positionExtrema := ruckig._profiles[1].positionExtrema();
AssertEquals_LREAL(0.13598633944686283614, positionExtrema.Tmax, 1E-9, message:='Profile[1] Tmax incorrect');
AssertEquals_LREAL(5.98711873384755755012, positionExtrema.Maximum, 1E-9, message:='Profile[1] maximum incorrect');
AssertEquals_LREAL(0.00000000000000000000, positionExtrema.Tmin, 1E-9, message:='Profile[1] Tmin incorrect');
AssertEquals_LREAL(-77.67370458831963730972, positionExtrema.Minimum, 1E-9, message:='Profile[1] minimum incorrect');

positionExtrema := ruckig._profiles[2].positionExtrema();
AssertEquals_LREAL(0.14901888909886754075, positionExtrema.Tmax, 1E-9, message:='Profile[2] Tmax incorrect');
AssertEquals_LREAL(92.98580498819549688960, positionExtrema.Maximum, 1E-9, message:='Profile[2] maximum incorrect');
AssertEquals_LREAL(0.00000000000000000000, positionExtrema.Tmin, 1E-9, message:='Profile[2] Tmin incorrect');
AssertEquals_LREAL(-11.76145133517785268396, positionExtrema.Minimum, 1E-9, message:='Profile[2] minimum incorrect');
   

TEST_FINISHED();
END_METHOD

METHOD Test_Trajectory_HasTargetVelocity_HasTargetAcceleration_41
VAR_INST
  ruckig : Struckig.Otg(0.001, 3) := (
  
    Synchronization := SynchronizationType.TimeSync,        
    MaxVelocity := [ 2000.00000000000000000000, 2000.00000000000000000000, 2000.00000000000000000000 ],
    MaxAcceleration := [ 20000.00000000000000000000, 20000.00000000000000000000, 20000.00000000000000000000 ],
    MaxJerk := [ 800000.00000000000000000000, 800000.00000000000000000000, 800000.00000000000000000000 ],
    CurrentPosition := [ 77.70133891525995295524, 7.01592092562633240505, 41.88398938907070601090 ],
    CurrentVelocity := [ -954.47536643469038608600, -572.16261829852851406031, 473.16402135503631143365 ],
    CurrentAcceleration := [ -2847.17654342300011194311, -1889.61698757276462856680, -3110.21768918452016805531 ],
    TargetPosition := [ 92.37579717709354554245, -14.04614057772144519731, -73.88361356505039623244 ],
    TargetVelocity := [ 519.95772801058456025203, 127.89327712966064609645, -380.91422286825297760515 ],
    TargetAcceleration := [ -890.64075852453197512659, 681.51569675393488978443, 390.99828361762297390669 ]
  );
  
  positionExtrema : Struckig.PositionExtremaDesc;
END_VAR
TEST('Trajectory_HasTargetVelocity_HasTargetAcceleration_41');

ruckig();

// Check total duration of profiles
AssertEquals_LREAL(Expected := 0.18543052523247699481, Actual := ruckig.Duration, DELTA := 1E-8, Message := 'Duration incorrect');

// Check duration for each phase
positionExtrema := ruckig._profiles[0].positionExtrema();
AssertEquals_LREAL(0.18543052523247699481, positionExtrema.Tmax, 1E-9, message:='Profile[0] Tmax incorrect');
AssertEquals_LREAL(92.37579717709354554245, positionExtrema.Maximum, 1E-9, message:='Profile[0] maximum incorrect');
AssertEquals_LREAL(0.07568410654937982041, positionExtrema.Tmin, 1E-9, message:='Profile[0] Tmin incorrect');
AssertEquals_LREAL(41.15768150995504015555, positionExtrema.Minimum, 1E-9, message:='Profile[0] minimum incorrect');

positionExtrema := ruckig._profiles[1].positionExtrema();
AssertEquals_LREAL(0.00000000000000000000, positionExtrema.Tmax, 1E-9, message:='Profile[1] Tmax incorrect');
AssertEquals_LREAL(7.01592092562633240505, positionExtrema.Maximum, 1E-9, message:='Profile[1] maximum incorrect');
AssertEquals_LREAL(0.16752625845292970497, positionExtrema.Tmin, 1E-9, message:='Profile[1] Tmin incorrect');
AssertEquals_LREAL(-15.47801998831725711625, positionExtrema.Minimum, 1E-9, message:='Profile[1] minimum incorrect');

positionExtrema := ruckig._profiles[2].positionExtrema();
AssertEquals_LREAL(0.02111222788851935261, positionExtrema.Tmax, 1E-9, message:='Profile[2] Tmax incorrect');
AssertEquals_LREAL(49.92568034606993876423, positionExtrema.Maximum, 1E-9, message:='Profile[2] maximum incorrect');
AssertEquals_LREAL(0.18543052523247699481, positionExtrema.Tmin, 1E-9, message:='Profile[2] Tmin incorrect');
AssertEquals_LREAL(-73.88361356505039623244, positionExtrema.Minimum, 1E-9, message:='Profile[2] minimum incorrect');
   

TEST_FINISHED();
END_METHOD

METHOD Test_Trajectory_HasTargetVelocity_HasTargetAcceleration_46
VAR_INST
  ruckig : Struckig.Otg(0.001, 3) := (
  
    Synchronization := SynchronizationType.TimeSync,        
    MaxVelocity := [ 2000.00000000000000000000, 2000.00000000000000000000, 2000.00000000000000000000 ],
    MaxAcceleration := [ 20000.00000000000000000000, 20000.00000000000000000000, 20000.00000000000000000000 ],
    MaxJerk := [ 800000.00000000000000000000, 800000.00000000000000000000, 800000.00000000000000000000 ],
    CurrentPosition := [ -81.70058267564624543411, -19.21897702137916041920, 94.53377990477645198553 ],
    CurrentVelocity := [ 791.96608977333426082623, 567.98007664216197554197, 949.19373974938935134560 ],
    CurrentAcceleration := [ -9852.41254141048739256803, -751.99368634466736693867, 3617.41551680202064744662 ],
    TargetPosition := [ 4.61526430014728816786, 47.19472748930556349478, -27.25527375543330776964 ],
    TargetVelocity := [ -365.39593288733976805815, -832.73312185042618693842, 15.48785727174674775597 ],
    TargetAcceleration := [ 393.54024330782590368472, -760.25458815149545444001, 23.06111995903222577908 ]
  );
  
  positionExtrema : Struckig.PositionExtremaDesc;
END_VAR
TEST('Trajectory_HasTargetVelocity_HasTargetAcceleration_46');

ruckig();

// Check total duration of profiles
AssertEquals_LREAL(Expected := 0.25941536116832880632, Actual := ruckig.Duration, DELTA := 1E-8, Message := 'Duration incorrect');

// Check duration for each phase
positionExtrema := ruckig._profiles[0].positionExtrema();
AssertEquals_LREAL(0.23392343586419403478, positionExtrema.Tmax, 1E-9, message:='Profile[0] Tmax incorrect');
AssertEquals_LREAL(11.84902844379517183881, positionExtrema.Maximum, 1E-9, message:='Profile[0] maximum incorrect');
AssertEquals_LREAL(0.00000000000000000000, positionExtrema.Tmin, 1E-9, message:='Profile[0] Tmin incorrect');
AssertEquals_LREAL(-81.70058267564624543411, positionExtrema.Minimum, 1E-9, message:='Profile[0] minimum incorrect');

positionExtrema := ruckig._profiles[1].positionExtrema();
AssertEquals_LREAL(0.19491405447314413824, positionExtrema.Tmax, 1E-9, message:='Profile[1] Tmax incorrect');
AssertEquals_LREAL(72.37093782213797510394, positionExtrema.Maximum, 1E-9, message:='Profile[1] maximum incorrect');
AssertEquals_LREAL(0.00000000000000000000, positionExtrema.Tmin, 1E-9, message:='Profile[1] Tmin incorrect');
AssertEquals_LREAL(-19.21897702137916041920, positionExtrema.Minimum, 1E-9, message:='Profile[1] minimum incorrect');

positionExtrema := ruckig._profiles[2].positionExtrema();
AssertEquals_LREAL(0.02952176939600252917, positionExtrema.Tmax, 1E-9, message:='Profile[2] Tmax incorrect');
AssertEquals_LREAL(120.70144362619019773319, positionExtrema.Maximum, 1E-9, message:='Profile[2] maximum incorrect');
AssertEquals_LREAL(0.25322160979530433655, positionExtrema.Tmin, 1E-9, message:='Profile[2] Tmin incorrect');
AssertEquals_LREAL(-27.31907826634350300310, positionExtrema.Minimum, 1E-9, message:='Profile[2] minimum incorrect');
   

TEST_FINISHED();
END_METHOD

METHOD Test_Trajectory_HasTargetVelocity_HasTargetAcceleration_47
VAR_INST
  ruckig : Struckig.Otg(0.001, 3) := (
  
    Synchronization := SynchronizationType.TimeSync,        
    MaxVelocity := [ 2000.00000000000000000000, 2000.00000000000000000000, 2000.00000000000000000000 ],
    MaxAcceleration := [ 20000.00000000000000000000, 20000.00000000000000000000, 20000.00000000000000000000 ],
    MaxJerk := [ 800000.00000000000000000000, 800000.00000000000000000000, 800000.00000000000000000000 ],
    CurrentPosition := [ 81.61368863479273727535, 18.81647567172932156154, -89.15971183512543518646 ],
    CurrentVelocity := [ 614.05723536338791745948, 343.05287387529847364931, -371.00163086153361291508 ],
    CurrentAcceleration := [ 2762.36060607538092881441, -8252.84383845068077789620, 1522.48694311787949118298 ],
    TargetPosition := [ 31.53792392446635517445, -13.15393306556988761713, -67.81554985684867631335 ],
    TargetVelocity := [ 927.36256285251761255495, -453.39442766394324735302, -734.53754957298599492788 ],
    TargetAcceleration := [ -810.42747656261008160072, 683.82844872197824770410, -296.63416710646515639382 ]
  );
  
  positionExtrema : Struckig.PositionExtremaDesc;
END_VAR
TEST('Trajectory_HasTargetVelocity_HasTargetAcceleration_47');

ruckig();

// Check total duration of profiles
AssertEquals_LREAL(Expected := 0.25287606970423076591, Actual := ruckig.Duration, DELTA := 1E-8, Message := 'Duration incorrect');

// Check duration for each phase
positionExtrema := ruckig._profiles[0].positionExtrema();
AssertEquals_LREAL(0.02845295075759422462, positionExtrema.Tmax, 1E-9, message:='Profile[0] Tmax incorrect');
AssertEquals_LREAL(97.13230269209392986340, positionExtrema.Maximum, 1E-9, message:='Profile[0] maximum incorrect');
AssertEquals_LREAL(0.22686303535852750390, positionExtrema.Tmin, 1E-9, message:='Profile[0] Tmin incorrect');
AssertEquals_LREAL(9.48720344289291794837, positionExtrema.Minimum, 1E-9, message:='Profile[0] minimum incorrect');

positionExtrema := ruckig._profiles[1].positionExtrema();
AssertEquals_LREAL(0.02241468542399701822, positionExtrema.Tmax, 1E-9, message:='Profile[1] Tmax incorrect');
AssertEquals_LREAL(23.03639977720293785524, positionExtrema.Maximum, 1E-9, message:='Profile[1] maximum incorrect');
AssertEquals_LREAL(0.25287606970423076591, positionExtrema.Tmin, 1E-9, message:='Profile[1] Tmin incorrect');
AssertEquals_LREAL(-13.15393306556988761713, positionExtrema.Minimum, 1E-9, message:='Profile[1] minimum incorrect');

positionExtrema := ruckig._profiles[2].positionExtrema();
AssertEquals_LREAL(0.20039624088411220337, positionExtrema.Tmax, 1E-9, message:='Profile[2] Tmax incorrect');
AssertEquals_LREAL(-46.06681198459425274905, positionExtrema.Maximum, 1E-9, message:='Profile[2] maximum incorrect');
AssertEquals_LREAL(0.03284040362274634473, positionExtrema.Tmin, 1E-9, message:='Profile[2] Tmin incorrect');
AssertEquals_LREAL(-95.92347928545005686374, positionExtrema.Minimum, 1E-9, message:='Profile[2] minimum incorrect');
   

TEST_FINISHED();
END_METHOD

METHOD Test_Trajectory_HasTargetVelocity_HasTargetAcceleration_48
VAR_INST
  ruckig : Struckig.Otg(0.001, 3) := (
  
    Synchronization := SynchronizationType.TimeSync,        
    MaxVelocity := [ 2000.00000000000000000000, 2000.00000000000000000000, 2000.00000000000000000000 ],
    MaxAcceleration := [ 20000.00000000000000000000, 20000.00000000000000000000, 20000.00000000000000000000 ],
    MaxJerk := [ 800000.00000000000000000000, 800000.00000000000000000000, 800000.00000000000000000000 ],
    CurrentPosition := [ -88.66208591478776668282, -31.58880789945652622919, 65.04291982806716987398 ],
    CurrentVelocity := [ 580.03497340359649570019, -746.36896556027750193607, 812.20588456619907447021 ],
    CurrentAcceleration := [ -6519.58462448879436124116, -9252.12079111587627266999, -5505.83185145304014440626 ],
    TargetPosition := [ -85.04127215306982634502, -92.28954144915404356198, -74.37698578032075147348 ],
    TargetVelocity := [ -365.82662455999411577068, -112.69189210154274860543, 154.77689249662125803297 ],
    TargetAcceleration := [ -682.87003825383567345852, -247.18670592987155032461, -122.60845320130738400621 ]
  );
  
  positionExtrema : Struckig.PositionExtremaDesc;
END_VAR
TEST('Trajectory_HasTargetVelocity_HasTargetAcceleration_48');

ruckig();

// Check total duration of profiles
AssertEquals_LREAL(Expected := 0.25037129752792702808, Actual := ruckig.Duration, DELTA := 1E-8, Message := 'Duration incorrect');

// Check duration for each phase
positionExtrema := ruckig._profiles[0].positionExtrema();
AssertEquals_LREAL(0.04415928948418586242, positionExtrema.Tmax, 1E-9, message:='Profile[0] Tmax incorrect');
AssertEquals_LREAL(-76.79539758143890537667, positionExtrema.Maximum, 1E-9, message:='Profile[0] maximum incorrect');
AssertEquals_LREAL(0.00000000000000000000, positionExtrema.Tmin, 1E-9, message:='Profile[0] Tmin incorrect');
AssertEquals_LREAL(-88.66208591478776668282, positionExtrema.Minimum, 1E-9, message:='Profile[0] minimum incorrect');

positionExtrema := ruckig._profiles[1].positionExtrema();
AssertEquals_LREAL(0.00000000000000000000, positionExtrema.Tmax, 1E-9, message:='Profile[1] Tmax incorrect');
AssertEquals_LREAL(-31.58880789945652622919, positionExtrema.Maximum, 1E-9, message:='Profile[1] maximum incorrect');
AssertEquals_LREAL(0.25037129752792697257, positionExtrema.Tmin, 1E-9, message:='Profile[1] Tmin incorrect');
AssertEquals_LREAL(-92.28954144915404356198, positionExtrema.Minimum, 1E-9, message:='Profile[1] minimum incorrect');

positionExtrema := ruckig._profiles[2].positionExtrema();
AssertEquals_LREAL(0.01811771018568369973, positionExtrema.Tmax, 1E-9, message:='Profile[2] Tmax incorrect');
AssertEquals_LREAL(78.06162686897538094399, positionExtrema.Maximum, 1E-9, message:='Profile[2] maximum incorrect');
AssertEquals_LREAL(0.23054659268189173216, positionExtrema.Tmin, 1E-9, message:='Profile[2] Tmin incorrect');
AssertEquals_LREAL(-76.43062116116439597135, positionExtrema.Minimum, 1E-9, message:='Profile[2] minimum incorrect');
   

TEST_FINISHED();
END_METHOD

METHOD Test_Trajectory_HasTargetVelocity_HasTargetAcceleration_51
VAR_INST
  ruckig : Struckig.Otg(0.001, 3) := (
  
    Synchronization := SynchronizationType.TimeSync,        
    MaxVelocity := [ 2000.00000000000000000000, 2000.00000000000000000000, 2000.00000000000000000000 ],
    MaxAcceleration := [ 20000.00000000000000000000, 20000.00000000000000000000, 20000.00000000000000000000 ],
    MaxJerk := [ 800000.00000000000000000000, 800000.00000000000000000000, 800000.00000000000000000000 ],
    CurrentPosition := [ 52.80919631150752024951, -81.68038555889982887948, 42.06917442755320735159 ],
    CurrentVelocity := [ -848.38044536898496517097, -694.53443230755419790512, -67.27027959540748724976 ],
    CurrentAcceleration := [ -7839.42279939661148091545, 2086.65454098016925854608, -1769.91408787331420171540 ],
    TargetPosition := [ 18.36498902426966139956, 7.18108207234031681310, -24.86667965964299753523 ],
    TargetVelocity := [ -484.52530887106502177630, -330.54249305132475456048, 184.78707869201707580942 ],
    TargetAcceleration := [ 34.47472473095945133537, 524.15868234202798703336, 659.72269096659351816925 ]
  );
  
  positionExtrema : Struckig.PositionExtremaDesc;
END_VAR
TEST('Trajectory_HasTargetVelocity_HasTargetAcceleration_51');

ruckig();

// Check total duration of profiles
AssertEquals_LREAL(Expected := 0.22814955969060143892, Actual := ruckig.Duration, DELTA := 1E-8, Message := 'Duration incorrect');

// Check duration for each phase
positionExtrema := ruckig._profiles[0].positionExtrema();
AssertEquals_LREAL(0.00000000000000000000, positionExtrema.Tmax, 1E-9, message:='Profile[0] Tmax incorrect');
AssertEquals_LREAL(52.80919631150752024951, positionExtrema.Maximum, 1E-9, message:='Profile[0] maximum incorrect');
AssertEquals_LREAL(0.06738171645932469755, positionExtrema.Tmin, 1E-9, message:='Profile[0] Tmin incorrect');
AssertEquals_LREAL(13.99608603958429142722, positionExtrema.Minimum, 1E-9, message:='Profile[0] minimum incorrect');

positionExtrema := ruckig._profiles[1].positionExtrema();
AssertEquals_LREAL(0.20249436133767390045, positionExtrema.Tmax, 1E-9, message:='Profile[1] Tmax incorrect');
AssertEquals_LREAL(13.58224981559266097975, positionExtrema.Maximum, 1E-9, message:='Profile[1] maximum incorrect');
AssertEquals_LREAL(0.02239168182377478805, positionExtrema.Tmin, 1E-9, message:='Profile[1] Tmin incorrect');
AssertEquals_LREAL(-95.21214742443424938756, positionExtrema.Minimum, 1E-9, message:='Profile[1] minimum incorrect');

positionExtrema := ruckig._profiles[2].positionExtrema();
AssertEquals_LREAL(0.00000000000000000000, positionExtrema.Tmax, 1E-9, message:='Profile[2] Tmax incorrect');
AssertEquals_LREAL(42.06917442755320735159, positionExtrema.Maximum, 1E-9, message:='Profile[2] maximum incorrect');
AssertEquals_LREAL(0.20746496504559683305, positionExtrema.Tmin, 1E-9, message:='Profile[2] Tmin incorrect');
AssertEquals_LREAL(-27.36779954300167716497, positionExtrema.Minimum, 1E-9, message:='Profile[2] minimum incorrect');
   

TEST_FINISHED();
END_METHOD

METHOD Test_Trajectory_HasTargetVelocity_HasTargetAcceleration_56
VAR_INST
  ruckig : Struckig.Otg(0.001, 3) := (
  
    Synchronization := SynchronizationType.TimeSync,        
    MaxVelocity := [ 2000.00000000000000000000, 2000.00000000000000000000, 2000.00000000000000000000 ],
    MaxAcceleration := [ 20000.00000000000000000000, 20000.00000000000000000000, 20000.00000000000000000000 ],
    MaxJerk := [ 800000.00000000000000000000, 800000.00000000000000000000, 800000.00000000000000000000 ],
    CurrentPosition := [ -75.10494070961726720270, -6.22395011546019816251, 35.64048680664691914899 ],
    CurrentVelocity := [ -825.41867748520257919154, -559.17669137031361970003, 331.05712850319173412572 ],
    CurrentAcceleration := [ -2748.49249899548522080295, -2734.78689775577458931366, 8828.96129221495357342064 ],
    TargetPosition := [ -88.93249178580995817356, 32.61549251092765189242, -4.33333209618611192582 ],
    TargetVelocity := [ -969.86803709259822880995, 219.52159207481986413768, 145.45315840784223837545 ],
    TargetAcceleration := [ 673.73439439858611876843, 589.54870253816602598818, 268.61037017006333371683 ]
  );
  
  positionExtrema : Struckig.PositionExtremaDesc;
END_VAR
TEST('Trajectory_HasTargetVelocity_HasTargetAcceleration_56');

ruckig();

// Check total duration of profiles
AssertEquals_LREAL(Expected := 0.22533279528439006945, Actual := ruckig.Duration, DELTA := 1E-8, Message := 'Duration incorrect');

// Check duration for each phase
positionExtrema := ruckig._profiles[0].positionExtrema();
AssertEquals_LREAL(0.13546282954524005437, positionExtrema.Tmax, 1E-9, message:='Profile[0] Tmax incorrect');
AssertEquals_LREAL(-60.83093977470542768060, positionExtrema.Maximum, 1E-9, message:='Profile[0] maximum incorrect');
AssertEquals_LREAL(0.08546282954524006548, positionExtrema.Tmin, 1E-9, message:='Profile[0] Tmin incorrect');
AssertEquals_LREAL(-97.18448406099201974939, positionExtrema.Minimum, 1E-9, message:='Profile[0] minimum incorrect');

positionExtrema := ruckig._profiles[1].positionExtrema();
AssertEquals_LREAL(0.22533279528439004169, positionExtrema.Tmax, 1E-9, message:='Profile[1] Tmax incorrect');
AssertEquals_LREAL(32.61549251092765189242, positionExtrema.Maximum, 1E-9, message:='Profile[1] maximum incorrect');
AssertEquals_LREAL(0.04813186201257521613, positionExtrema.Tmin, 1E-9, message:='Profile[1] Tmin incorrect');
AssertEquals_LREAL(-22.45997635018479243740, positionExtrema.Minimum, 1E-9, message:='Profile[1] minimum incorrect');

positionExtrema := ruckig._profiles[2].positionExtrema();
AssertEquals_LREAL(0.04893648758049205100, positionExtrema.Tmax, 1E-9, message:='Profile[2] Tmax incorrect');
AssertEquals_LREAL(47.07359821757206930215, positionExtrema.Maximum, 1E-9, message:='Profile[2] maximum incorrect');
AssertEquals_LREAL(0.20659644161609555524, positionExtrema.Tmin, 1E-9, message:='Profile[2] Tmin incorrect');
AssertEquals_LREAL(-6.13445732070238047839, positionExtrema.Minimum, 1E-9, message:='Profile[2] minimum incorrect');
   

TEST_FINISHED();
END_METHOD

METHOD Test_Trajectory_HasTargetVelocity_HasTargetAcceleration_60
VAR_INST
  ruckig : Struckig.Otg(0.001, 3) := (
  
    Synchronization := SynchronizationType.TimeSync,        
    MaxVelocity := [ 2000.00000000000000000000, 2000.00000000000000000000, 2000.00000000000000000000 ],
    MaxAcceleration := [ 20000.00000000000000000000, 20000.00000000000000000000, 20000.00000000000000000000 ],
    MaxJerk := [ 800000.00000000000000000000, 800000.00000000000000000000, 800000.00000000000000000000 ],
    CurrentPosition := [ -82.30425131320278353542, 95.77277574475397159404, -0.37873053404373990816 ],
    CurrentVelocity := [ 209.81667767709768668283, 666.24835564548857291811, -156.12978395261052355636 ],
    CurrentAcceleration := [ 554.62083613543836690951, 1781.55274365866716834716, -2304.74829583103382901754 ],
    TargetPosition := [ 78.56604956044506593571, -99.70839917358892989796, -88.26279812419441839211 ],
    TargetVelocity := [ 182.35588906091311400814, 216.59536701599199659540, -100.01197301996137412061 ],
    TargetAcceleration := [ 165.30880475002527418837, -915.29760737648621216067, 984.89234990536533587147 ]
  );
  
  positionExtrema : Struckig.PositionExtremaDesc;
END_VAR
TEST('Trajectory_HasTargetVelocity_HasTargetAcceleration_60');

ruckig();

// Check total duration of profiles
AssertEquals_LREAL(Expected := 0.28418047012119368455, Actual := ruckig.Duration, DELTA := 1E-8, Message := 'Duration incorrect');

// Check duration for each phase
positionExtrema := ruckig._profiles[0].positionExtrema();
AssertEquals_LREAL(0.28418047012119368455, positionExtrema.Tmax, 1E-9, message:='Profile[0] Tmax incorrect');
AssertEquals_LREAL(78.56604956044506593571, positionExtrema.Maximum, 1E-9, message:='Profile[0] maximum incorrect');
AssertEquals_LREAL(0.00000000000000000000, positionExtrema.Tmin, 1E-9, message:='Profile[0] Tmin incorrect');
AssertEquals_LREAL(-82.30425131320278353542, positionExtrema.Minimum, 1E-9, message:='Profile[0] minimum incorrect');

positionExtrema := ruckig._profiles[1].positionExtrema();
AssertEquals_LREAL(0.02722694092957333306, positionExtrema.Tmax, 1E-9, message:='Profile[1] Tmax incorrect');
AssertEquals_LREAL(111.88188475863630344520, positionExtrema.Maximum, 1E-9, message:='Profile[1] maximum incorrect');
AssertEquals_LREAL(0.25973833461914580534, positionExtrema.Tmin, 1E-9, message:='Profile[1] Tmin incorrect');
AssertEquals_LREAL(-103.32890392255741573990, positionExtrema.Minimum, 1E-9, message:='Profile[1] minimum incorrect');

positionExtrema := ruckig._profiles[2].positionExtrema();
AssertEquals_LREAL(0.00000000000000000000, positionExtrema.Tmax, 1E-9, message:='Profile[2] Tmax incorrect');
AssertEquals_LREAL(-0.37873053404373990816, positionExtrema.Maximum, 1E-9, message:='Profile[2] maximum incorrect');
AssertEquals_LREAL(0.28418047012119368455, positionExtrema.Tmin, 1E-9, message:='Profile[2] Tmin incorrect');
AssertEquals_LREAL(-88.26279812419441839211, positionExtrema.Minimum, 1E-9, message:='Profile[2] minimum incorrect');
   

TEST_FINISHED();
END_METHOD

METHOD Test_Trajectory_HasTargetVelocity_HasTargetAcceleration_61
VAR_INST
  ruckig : Struckig.Otg(0.001, 3) := (
  
    Synchronization := SynchronizationType.TimeSync,        
    MaxVelocity := [ 2000.00000000000000000000, 2000.00000000000000000000, 2000.00000000000000000000 ],
    MaxAcceleration := [ 20000.00000000000000000000, 20000.00000000000000000000, 20000.00000000000000000000 ],
    MaxJerk := [ 800000.00000000000000000000, 800000.00000000000000000000, 800000.00000000000000000000 ],
    CurrentPosition := [ 69.02958196301639759440, -13.39780118806328346182, -96.66107573544628905893 ],
    CurrentVelocity := [ 100.84225227141041614232, -40.44627894454811212199, 363.36834103503497317433 ],
    CurrentAcceleration := [ -7135.55942272971151396632, -622.60760459453013027087, 1671.34292984182866348419 ],
    TargetPosition := [ -16.84074689714994121914, -92.09682308688789476037, -87.06215904519353898650 ],
    TargetVelocity := [ 537.25106843782555188227, -935.18562117857493376505, -396.85249080038204283483 ],
    TargetAcceleration := [ -310.44042758873558796040, -501.02391325450025760802, -57.28028759093501776078 ]
  );
  
  positionExtrema : Struckig.PositionExtremaDesc;
END_VAR
TEST('Trajectory_HasTargetVelocity_HasTargetAcceleration_61');

ruckig();

// Check total duration of profiles
AssertEquals_LREAL(Expected := 0.19429164835544748824, Actual := ruckig.Duration, DELTA := 1E-8, Message := 'Duration incorrect');

// Check duration for each phase
positionExtrema := ruckig._profiles[0].positionExtrema();
AssertEquals_LREAL(0.00929214609675180735, positionExtrema.Tmax, 1E-9, message:='Profile[0] Tmax incorrect');
AssertEquals_LREAL(69.55159049131329140891, positionExtrema.Maximum, 1E-9, message:='Profile[0] maximum incorrect');
AssertEquals_LREAL(0.16890359782096156516, positionExtrema.Tmin, 1E-9, message:='Profile[0] Tmin incorrect');
AssertEquals_LREAL(-28.39869225356863324805, positionExtrema.Minimum, 1E-9, message:='Profile[0] minimum incorrect');

positionExtrema := ruckig._profiles[1].positionExtrema();
AssertEquals_LREAL(0.00000000000000000000, positionExtrema.Tmax, 1E-9, message:='Profile[1] Tmax incorrect');
AssertEquals_LREAL(-13.39780118806328346182, positionExtrema.Maximum, 1E-9, message:='Profile[1] maximum incorrect');
AssertEquals_LREAL(0.19429164835544748824, positionExtrema.Tmin, 1E-9, message:='Profile[1] Tmin incorrect');
AssertEquals_LREAL(-92.09682308688789476037, positionExtrema.Minimum, 1E-9, message:='Profile[1] minimum incorrect');

positionExtrema := ruckig._profiles[2].positionExtrema();
AssertEquals_LREAL(0.15958331587242960414, positionExtrema.Tmax, 1E-9, message:='Profile[2] Tmax incorrect');
AssertEquals_LREAL(-78.59507311744690127853, positionExtrema.Maximum, 1E-9, message:='Profile[2] maximum incorrect');
AssertEquals_LREAL(0.00000000000000000000, positionExtrema.Tmin, 1E-9, message:='Profile[2] Tmin incorrect');
AssertEquals_LREAL(-96.66107573544628905893, positionExtrema.Minimum, 1E-9, message:='Profile[2] minimum incorrect');
   

TEST_FINISHED();
END_METHOD

METHOD Test_Trajectory_HasTargetVelocity_HasTargetAcceleration_66
VAR_INST
  ruckig : Struckig.Otg(0.001, 3) := (
  
    Synchronization := SynchronizationType.TimeSync,        
    MaxVelocity := [ 2000.00000000000000000000, 2000.00000000000000000000, 2000.00000000000000000000 ],
    MaxAcceleration := [ 20000.00000000000000000000, 20000.00000000000000000000, 20000.00000000000000000000 ],
    MaxJerk := [ 800000.00000000000000000000, 800000.00000000000000000000, 800000.00000000000000000000 ],
    CurrentPosition := [ -48.80987185641822634352, 18.04364910313265113473, -24.74266082352920648191 ],
    CurrentVelocity := [ 988.42910759631240580347, -768.41448219800986407790, -207.75563249912386254437 ],
    CurrentAcceleration := [ 3735.71066306482680374756, -9295.98081225150599493645, 5866.28306601172880618833 ],
    TargetPosition := [ -12.17413972252995790768, 39.46835789725682275275, -82.53347662682273266910 ],
    TargetVelocity := [ 196.90336440418968777522, 718.33687283187941829965, -527.62167018153525077651 ],
    TargetAcceleration := [ -832.60782943610661277489, 502.29848616551748818893, 413.82241950646152872650 ]
  );
  
  positionExtrema : Struckig.PositionExtremaDesc;
END_VAR
TEST('Trajectory_HasTargetVelocity_HasTargetAcceleration_66');

ruckig();

// Check total duration of profiles
AssertEquals_LREAL(Expected := 0.15504630751390929833, Actual := ruckig.Duration, DELTA := 1E-8, Message := 'Duration incorrect');

// Check duration for each phase
positionExtrema := ruckig._profiles[0].positionExtrema();
AssertEquals_LREAL(0.06757881268766546823, positionExtrema.Tmax, 1E-9, message:='Profile[0] Tmax incorrect');
AssertEquals_LREAL(-7.34951569385982939053, positionExtrema.Maximum, 1E-9, message:='Profile[0] maximum incorrect');
AssertEquals_LREAL(0.00000000000000000000, positionExtrema.Tmin, 1E-9, message:='Profile[0] Tmin incorrect');
AssertEquals_LREAL(-48.80987185641822634352, positionExtrema.Minimum, 1E-9, message:='Profile[0] minimum incorrect');

positionExtrema := ruckig._profiles[1].positionExtrema();
AssertEquals_LREAL(0.15504630751390929833, positionExtrema.Tmax, 1E-9, message:='Profile[1] Tmax incorrect');
AssertEquals_LREAL(39.46835789725682275275, positionExtrema.Maximum, 1E-9, message:='Profile[1] maximum incorrect');
AssertEquals_LREAL(0.03661997601531438024, positionExtrema.Tmin, 1E-9, message:='Profile[1] Tmin incorrect');
AssertEquals_LREAL(-9.78096891406795521107, positionExtrema.Minimum, 1E-9, message:='Profile[1] minimum incorrect');

positionExtrema := ruckig._profiles[2].positionExtrema();
AssertEquals_LREAL(0.00000000000000000000, positionExtrema.Tmax, 1E-9, message:='Profile[2] Tmax incorrect');
AssertEquals_LREAL(-24.74266082352920648191, positionExtrema.Maximum, 1E-9, message:='Profile[2] maximum incorrect');
AssertEquals_LREAL(0.15504630751390929833, positionExtrema.Tmin, 1E-9, message:='Profile[2] Tmin incorrect');
AssertEquals_LREAL(-82.53347662682273266910, positionExtrema.Minimum, 1E-9, message:='Profile[2] minimum incorrect');
   

TEST_FINISHED();
END_METHOD

METHOD Test_Trajectory_HasTargetVelocity_HasTargetAcceleration_70
VAR_INST
  ruckig : Struckig.Otg(0.001, 3) := (
  
    Synchronization := SynchronizationType.TimeSync,        
    MaxVelocity := [ 2000.00000000000000000000, 2000.00000000000000000000, 2000.00000000000000000000 ],
    MaxAcceleration := [ 20000.00000000000000000000, 20000.00000000000000000000, 20000.00000000000000000000 ],
    MaxJerk := [ 800000.00000000000000000000, 800000.00000000000000000000, 800000.00000000000000000000 ],
    CurrentPosition := [ -92.33184858939047501281, 71.73781926022004995502, -55.27032026177170109804 ],
    CurrentVelocity := [ -952.87828015244156176777, -234.88833123485505893768, 123.27287252024666486250 ],
    CurrentAcceleration := [ -7266.87319497806674917229, -1917.48167665642540669069, -9579.01136324118306220043 ],
    TargetPosition := [ -64.62381428735777433303, 58.03768693667834099870, 63.08437907080863737974 ],
    TargetVelocity := [ 812.70256182329512739670, -863.39780178803880517080, -492.22548367060147711527 ],
    TargetAcceleration := [ 53.46404855095147468091, -729.77327604858464837889, -373.83030360848226791859 ]
  );
  
  positionExtrema : Struckig.PositionExtremaDesc;
END_VAR
TEST('Trajectory_HasTargetVelocity_HasTargetAcceleration_70');

ruckig();

// Check total duration of profiles
AssertEquals_LREAL(Expected := 0.22013991649512543169, Actual := ruckig.Duration, DELTA := 1E-8, Message := 'Duration incorrect');

// Check duration for each phase
positionExtrema := ruckig._profiles[0].positionExtrema();
AssertEquals_LREAL(0.22013991649512543169, positionExtrema.Tmax, 1E-9, message:='Profile[0] Tmax incorrect');
AssertEquals_LREAL(-64.62381428735777433303, positionExtrema.Maximum, 1E-9, message:='Profile[0] maximum incorrect');
AssertEquals_LREAL(0.08266151031223724355, positionExtrema.Tmin, 1E-9, message:='Profile[0] Tmin incorrect');
AssertEquals_LREAL(-135.90053229571682891219, positionExtrema.Minimum, 1E-9, message:='Profile[0] minimum incorrect');

positionExtrema := ruckig._profiles[1].positionExtrema();
AssertEquals_LREAL(0.16474949862477941687, positionExtrema.Tmax, 1E-9, message:='Profile[1] Tmax incorrect');
AssertEquals_LREAL(86.19544571063090643293, positionExtrema.Maximum, 1E-9, message:='Profile[1] maximum incorrect');
AssertEquals_LREAL(0.22013991649512543169, positionExtrema.Tmin, 1E-9, message:='Profile[1] Tmin incorrect');
AssertEquals_LREAL(58.03768693667834099870, positionExtrema.Minimum, 1E-9, message:='Profile[1] minimum incorrect');

positionExtrema := ruckig._profiles[2].positionExtrema();
AssertEquals_LREAL(0.19560720437463602339, positionExtrema.Tmax, 1E-9, message:='Profile[2] Tmax incorrect');
AssertEquals_LREAL(73.07882819675037922025, positionExtrema.Maximum, 1E-9, message:='Profile[2] maximum incorrect');
AssertEquals_LREAL(0.00000000000000000000, positionExtrema.Tmin, 1E-9, message:='Profile[2] Tmin incorrect');
AssertEquals_LREAL(-55.27032026177170109804, positionExtrema.Minimum, 1E-9, message:='Profile[2] minimum incorrect');
   

TEST_FINISHED();
END_METHOD

END_FUNCTION_BLOCK

// ---- POUs/PropagateTest.TcPOU
FUNCTION_BLOCK PropagateTest EXTENDS TcUnit.FB_TestSuite

Test_AutoPropagate();
Test_ManualPropagate();
Test_NoPropagate();

METHOD Test_AutoPropagate
VAR_INST
  ruckig : Struckig.Otg(0.001, 3) := (
  
    Synchronization := SynchronizationType.TimeSync,        
    MaxVelocity := [ 2000, 2000, 2000 ],
    MaxAcceleration := [ 20000, 20000, 20000 ],
    MaxJerk := [ 8000, 80000, 800000 ],
    CurrentPosition := [ 0,0,0  ],
    CurrentVelocity := [ 0,0,0 ],
    CurrentAcceleration := [ 0,0,0 ],
    TargetPosition := [ 1, 10, 100 ],
    TargetVelocity := [ 0,0,0 ],
    TargetAcceleration := [ 0,0,0 ]
  );
  
  StartPosition, StartVelocity, StartAcceleration : ARRAY[0..ParameterList.MaxDoFs] OF LREAL; // Current state
  NewPosition, NewVelocity, NewAcceleration : ARRAY[0..ParameterList.MaxDoFs] OF LREAL; // Current state  
END_VAR
TEST('Test_AutoPropagate');

StartPosition := ruckig.CurrentPosition;
StartVelocity := ruckig.CurrentVelocity;
StartAcceleration := ruckig.CurrentAcceleration;

ruckig();
AssertTrue(0 = ruckig.CurrentPosition[0], Message:=''); 

NewPosition := ruckig.NewPosition;
NewVelocity := ruckig.NewVelocity;
NewAcceleration := ruckig.NewAcceleration;

ruckig(EnableAutoPropagate := TRUE);

AssertTrue(0 <> ruckig.CurrentPosition[0], Message:=''); 
AssertArrayEquals_LREAL(Expecteds:=NewPosition, Actuals:=ruckig.CurrentPosition, Delta:=1E-6, Message:='');
AssertArrayEquals_LREAL(Expecteds:=NewVelocity, Actuals:=ruckig.CurrentVelocity, Delta:=1E-6, Message:='');
AssertArrayEquals_LREAL(Expecteds:=NewAcceleration, Actuals:=ruckig.CurrentAcceleration, Delta:=1E-6, Message:='');

TEST_FINISHED();
END_METHOD

METHOD Test_ManualPropagate
VAR_INST
  ruckig : Struckig.Otg(0.001, 3) := (
  
    Synchronization := SynchronizationType.TimeSync,        
    MaxVelocity := [ 2000, 2000, 2000 ],
    MaxAcceleration := [ 20000, 20000, 20000 ],
    MaxJerk := [ 8000, 80000, 800000 ],
    CurrentPosition := [ 0,0,0  ],
    CurrentVelocity := [ 0,0,0 ],
    CurrentAcceleration := [ 0,0,0 ],
    TargetPosition := [ 1, 10, 100 ],
    TargetVelocity := [ 0,0,0 ],
    TargetAcceleration := [ 0,0,0 ]
  );
  
  StartPosition, StartVelocity, StartAcceleration : ARRAY[0..ParameterList.MaxDoFs] OF LREAL; // Current state
  NewPosition, NewVelocity, NewAcceleration : ARRAY[0..ParameterList.MaxDoFs] OF LREAL; // Current state  
END_VAR
TEST('Test_ManualPropagate');

StartPosition := ruckig.CurrentPosition;
StartVelocity := ruckig.CurrentVelocity;
StartAcceleration := ruckig.CurrentAcceleration;

ruckig();
AssertTrue(0 = ruckig.CurrentPosition[0], Message:=''); 

NewPosition := ruckig.NewPosition;
NewVelocity := ruckig.NewVelocity;
NewAcceleration := ruckig.NewAcceleration;

ruckig.PassOutputToInput();

AssertTrue(0 <> ruckig.CurrentPosition[0], Message:=''); 
AssertArrayEquals_LREAL(Expecteds:=NewPosition, Actuals:=ruckig.CurrentPosition, Delta:=1E-6, Message:='');
AssertArrayEquals_LREAL(Expecteds:=NewVelocity, Actuals:=ruckig.CurrentVelocity, Delta:=1E-6, Message:='');
AssertArrayEquals_LREAL(Expecteds:=NewAcceleration, Actuals:=ruckig.CurrentAcceleration, Delta:=1E-6, Message:='');

TEST_FINISHED();
END_METHOD

METHOD Test_NoPropagate
VAR_INST
  ruckig : Struckig.Otg(0.001, 3) := (
  
    Synchronization := SynchronizationType.TimeSync,        
    MaxVelocity := [ 2000, 2000, 2000 ],
    MaxAcceleration := [ 20000, 20000, 20000 ],
    MaxJerk := [ 8000, 80000, 800000 ],
    CurrentPosition := [ 0,0,0  ],
    CurrentVelocity := [ 0,0,0 ],
    CurrentAcceleration := [ 0,0,0 ],
    TargetPosition := [ 1, 10, 100 ],
    TargetVelocity := [ 0,0,0 ],
    TargetAcceleration := [ 0,0,0 ]
  );
  
  StartPosition, StartVelocity, StartAcceleration : ARRAY[0..ParameterList.MaxDoFs] OF LREAL; // Current state
  NewPosition, NewVelocity, NewAcceleration : ARRAY[0..ParameterList.MaxDoFs] OF LREAL; // Current state  
END_VAR
TEST('Test_NoPropagate');

StartPosition := ruckig.CurrentPosition;
StartVelocity := ruckig.CurrentVelocity;
StartAcceleration := ruckig.CurrentAcceleration;

AssertArrayEquals_LREAL(Expecteds:=StartPosition, Actuals:=ruckig.CurrentPosition, Delta:=1E-6, Message:='');
AssertArrayEquals_LREAL(Expecteds:=StartVelocity, Actuals:=ruckig.CurrentVelocity, Delta:=1E-6, Message:='');
AssertArrayEquals_LREAL(Expecteds:=StartAcceleration, Actuals:=ruckig.CurrentAcceleration, Delta:=1E-6, Message:='');

ruckig();

AssertArrayEquals_LREAL(Expecteds:=StartPosition, Actuals:=ruckig.CurrentPosition, Delta:=1E-6, Message:='');
AssertArrayEquals_LREAL(Expecteds:=StartVelocity, Actuals:=ruckig.CurrentVelocity, Delta:=1E-6, Message:='');
AssertArrayEquals_LREAL(Expecteds:=StartAcceleration, Actuals:=ruckig.CurrentAcceleration, Delta:=1E-6, Message:='');

TEST_FINISHED();
END_METHOD

END_FUNCTION_BLOCK
